(* PLC project drill, Dassault Systèmes ControlBuild 2024x Refresh1 *)
(* stored: creationDateTime 2024-03-18T15:45:01-01:00 *)

FUNCTION_BLOCK clampingfunction
  VAR_INPUT
    acknowledgePB : BOOL := false;
    releasing : BOOL := false;
    clamping : BOOL := false;
    rightUnlocked : BOOL := false;
    rightLocked : BOOL := false;
    leftUnlocked : BOOL := false;
    leftLocked : BOOL := false;
    rightFault : BOOL := false;
    leftFault : BOOL := false;
  END_VAR
  VAR_IN_OUT
    clampingDuration : INT := 0;
    releasingDuration : INT := 0;
  END_VAR
  VAR_OUTPUT
    clampingOK : BOOL := false;
    releasingOK : BOOL := false;
    clampingFault : INT := 0;
    rightLocking : BOOL := false;
    leftLocking : BOOL := false;
  END_VAR


ACTION C_source_code:

END_ACTION
END_FUNCTION_BLOCK

FUNCTION_BLOCK actions
  VAR_INPUT
    autoMode : BOOL := false;
    manualMode : BOOL := false;
    autoFwdCmd : BOOL := false;
    autoBwdCmd : BOOL := false;
    autoHSCmd : BOOL := false;
    autoLSCmd : BOOL := false;
    forwardPB : BOOL := false;
    backwardPB : BOOL := false;
    highSpeedPB : BOOL := false;
    lowSpeedPB : BOOL := false;
    stopPB : BOOL := false;
    generalFault : BOOL := false;
    autoWorkCmd : Unknown := ();
    valveWorkPB : Unknown := ();
  END_VAR
  VAR_OUTPUT
    forwardCmd : BOOL := false;
    backwardCmd : BOOL := false;
    highSpeedCmd : BOOL := false;
    lowSpeedCmd : BOOL := false;
    workCmd : BOOL := false;
  END_VAR


ACTION C_source_code:

END_ACTION
END_FUNCTION_BLOCK

FUNCTION_BLOCK faults1
  VAR_INPUT
    forwardCmd : BOOL := false;
    backwardCmd : BOOL := false;
    highSpeedCmd : BOOL := false;
    lowSpeedCmd : BOOL := false;
    thermalFB : BOOL := false;
    forwardFB : BOOL := false;
    backwardFB : BOOL := false;
    highSpeedFB : BOOL := false;
    lowSpeedFB : BOOL := false;
    acknowledgePB : BOOL := false;
    outletSensor : Unknown := ();
    inletSensor : Unknown := ();
    workCmd : Unknown := ();
  END_VAR
  VAR_IN_OUT
    thermalFault : BOOL := false;
    forwardFBFault : BOOL := false;
    backwardFBFault : BOOL := false;
  END_VAR
  VAR_OUTPUT
    generalFault : BOOL := false;
  END_VAR


ACTION C_source_code:

END_ACTION
END_FUNCTION_BLOCK

PROGRAM cmdofjack
  VAR_INPUT
    autoMode : BOOL := false;
    manualMode : BOOL := false;
    autoWorkCmd : BOOL := false;
    valveWorkPB : BOOL := false;
    outletSensor : BOOL := false;
    inletSensor : BOOL := false;
    acknowledgePB : BOOL := false;
  END_VAR
  VAR_OUTPUT
    workCmd : BOOL := false;
    generalFault : BOOL := false;
  END_VAR

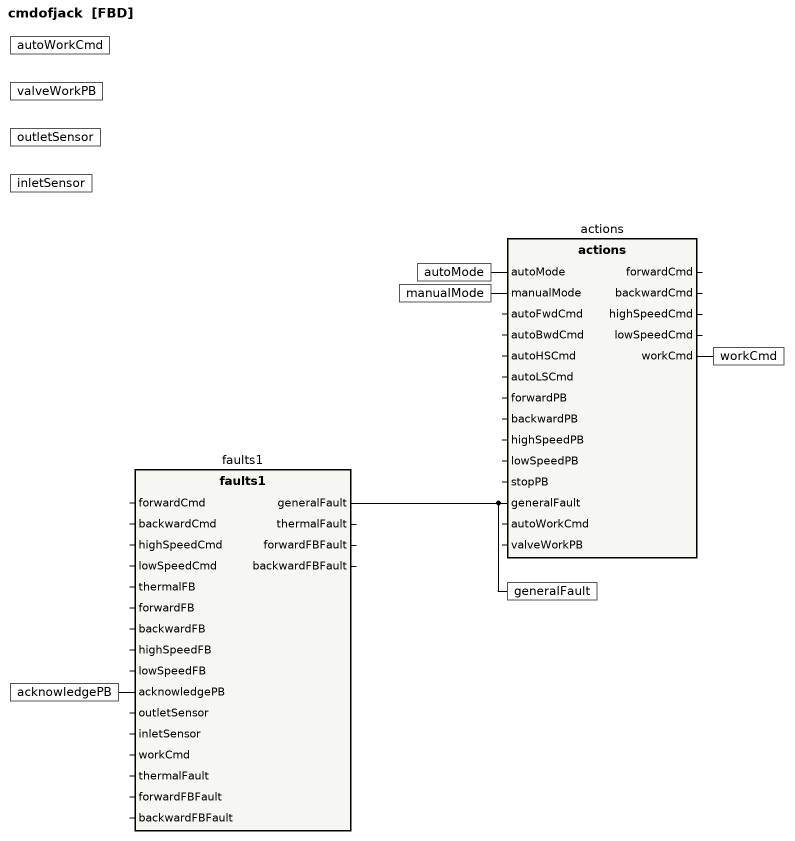
(* FBD diagram, written out as Structured Text *)
faults1(acknowledgePB := acknowledgePB);
actions(autoMode := autoMode, manualMode := manualMode, generalFault := faults1.generalFault);
workCmd := actions.workCmd;
generalFault := faults1.generalFault;
(* drawn but not wired to any output: autoWorkCmd, valveWorkPB, outletSensor, inletSensor *)
END_PROGRAM

FUNCTION_BLOCK jack
  VAR_INPUT
    energy : BOOL := false;
    cmdSupply : BOOL := false;
    sensorSupply : BOOL := false;
    valveWork : BOOL := false;
  END_VAR
  VAR_IN_OUT
    slidePosition : INT := 0;
    pipeWork : BOOL := false;
    pipeRest : BOOL := false;
    increment : REAL := 0.0;
    outletSensorLogic : BOOL := false;
    inletSensorLogic : BOOL := false;
    rodLength : REAL := 0.0;
    time2extend : REAL := 0.0;
    d_locking : BOOL := false;
    v_d_locking : REAL := 0.0;
    d_inletSensor : BOOL := false;
    v_d_inletSensor : BOOL := false;
    d_outletSensor : BOOL := false;
    v_d_outletSensor : BOOL := false;
  END_VAR
  VAR_OUTPUT
    outletSensor : BOOL := false;
    inletSensor : BOOL := false;
    rodPosition : REAL := 0.0;
    rodPercent : REAL := 0.0;
    incrementValue : REAL := 0.0;
  END_VAR


ACTION C_source_code:

END_ACTION
END_FUNCTION_BLOCK

FUNCTION_BLOCK backwardpb
  VAR_IN_OUT
    action : BOOL := false;
    timeCounter : REAL := 0.0;
    pulseDuration : REAL := 0.0;
    PBLogic : BOOL := false;
  END_VAR
  VAR_OUTPUT
    PB : BOOL := false;
  END_VAR


ACTION C_source_code:

END_ACTION
END_FUNCTION_BLOCK

FUNCTION_BLOCK forwardpb
  VAR_IN_OUT
    action : BOOL := false;
    timeCounter : REAL := 0.0;
    pulseDuration : REAL := 0.0;
    PBLogic : BOOL := false;
  END_VAR
  VAR_OUTPUT
    PB : BOOL := false;
  END_VAR


ACTION C_source_code:

END_ACTION
END_FUNCTION_BLOCK

FUNCTION_BLOCK speedswitch
  VAR_IN_OUT
    leftPosition : BOOL := false;
    rightPosition : BOOL := false;
  END_VAR
  VAR_OUTPUT
    leftVariable : BOOL := false;
    rightVariable : BOOL := false;
  END_VAR


ACTION C_source_code:

END_ACTION
END_FUNCTION_BLOCK

FUNCTION_BLOCK stoppb
  VAR_IN_OUT
    action : BOOL := false;
    timeCounter : REAL := 0.0;
    pulseDuration : REAL := 0.0;
    PBLogic : BOOL := false;
  END_VAR
  VAR_OUTPUT
    PB : BOOL := false;
  END_VAR


ACTION C_source_code:

END_ACTION
END_FUNCTION_BLOCK

PROGRAM panel1
  VAR_OUTPUT
    forwardPB : BOOL := false;
    backwardPB : BOOL := false;
    highSpeedPB : BOOL := false;
    lowSpeedPB : BOOL := false;
    stopPB : BOOL := false;
    valveWorkPB : BOOL := false;
  END_VAR

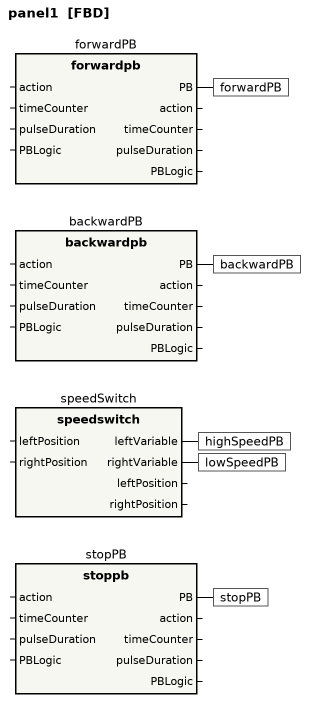
(* FBD diagram, written out as Structured Text *)
forwardPB();
forwardPB := forwardPB.PB;
backwardPB();
backwardPB := backwardPB.PB;
speedSwitch();
highSpeedPB := speedSwitch.leftVariable;
lowSpeedPB := speedSwitch.rightVariable;
stopPB();
stopPB := stopPB.PB;
END_PROGRAM

PROGRAM leftjack
  VAR_INPUT
    acknowledgePB : BOOL := false;
    autoMode : BOOL := false;
    manualMode : BOOL := false;
    autoWorkCmd : BOOL := false;
  END_VAR
  VAR_OUTPUT
    generalFault : BOOL := false;
    inletSensor : BOOL := false;
    outletSensor : BOOL := false;
    rodPosition : REAL := 0.0;
    rodPercent : REAL := 0.0;
    incrementValue : REAL := 0.0;
  END_VAR

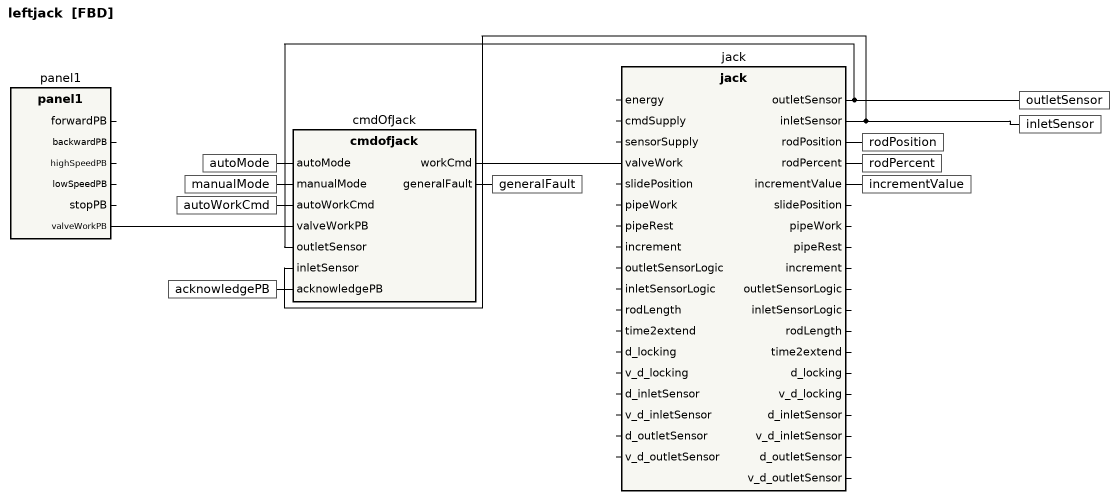
(* FBD diagram, written out as Structured Text *)
panel1();
jack(valveWork := cmdOfJack.workCmd);
cmdOfJack(autoMode := autoMode, manualMode := manualMode, autoWorkCmd := autoWorkCmd, valveWorkPB := panel1.valveWorkPB, outletSensor := jack.outletSensor, inletSensor := jack.inletSensor, acknowledgePB := acknowledgePB);
generalFault := cmdOfJack.generalFault;
inletSensor := jack.inletSensor;
outletSensor := jack.outletSensor;
rodPosition := jack.rodPosition;
rodPercent := jack.rodPercent;
incrementValue := jack.incrementValue;
END_PROGRAM

PROGRAM rightjack
  VAR_INPUT
    acknowledgePB : BOOL := false;
    autoMode : BOOL := false;
    manualMode : BOOL := false;
    autoWorkCmd : BOOL := false;
  END_VAR
  VAR_OUTPUT
    generalFault : BOOL := false;
    inletSensor : BOOL := false;
    outletSensor : BOOL := false;
    rodPosition : REAL := 0.0;
    rodPercent : REAL := 0.0;
    incrementValue : REAL := 0.0;
  END_VAR

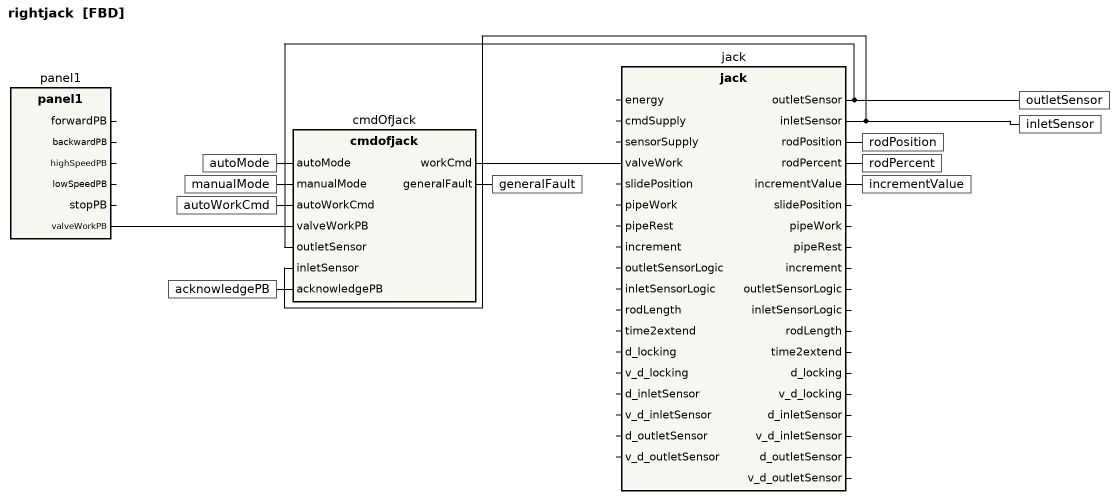
(* FBD diagram, written out as Structured Text *)
panel1();
jack(valveWork := cmdOfJack.workCmd);
cmdOfJack(autoMode := autoMode, manualMode := manualMode, autoWorkCmd := autoWorkCmd, valveWorkPB := panel1.valveWorkPB, outletSensor := jack.outletSensor, inletSensor := jack.inletSensor, acknowledgePB := acknowledgePB);
generalFault := cmdOfJack.generalFault;
inletSensor := jack.inletSensor;
outletSensor := jack.outletSensor;
rodPosition := jack.rodPosition;
rodPercent := jack.rodPercent;
incrementValue := jack.incrementValue;
END_PROGRAM

PROGRAM clamping
  VAR_INPUT
    acknowledgePB : BOOL := false;
    autoMode : BOOL := false;
    manualMode : BOOL := false;
    releasing : BOOL := false;
    clamping : BOOL := false;
  END_VAR
  VAR_OUTPUT
    clampingOK : BOOL := false;
    releasingOK : BOOL := false;
    clampingFault : INT := 0;
  END_VAR

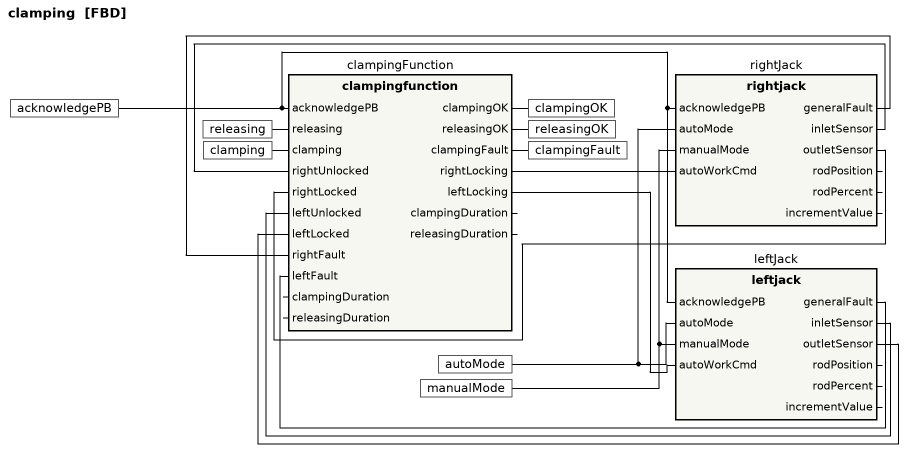
(* FBD diagram, written out as Structured Text *)
rightJack(acknowledgePB := acknowledgePB, autoMode := autoMode, manualMode := manualMode, autoWorkCmd := clampingFunction.rightLocking);
leftJack(acknowledgePB := acknowledgePB, autoMode := autoMode, manualMode := manualMode, autoWorkCmd := clampingFunction.leftLocking);
clampingFunction(acknowledgePB := acknowledgePB, releasing := releasing, clamping := clamping, rightUnlocked := rightJack.inletSensor, rightLocked := rightJack.outletSensor, leftUnlocked := leftJack.inletSensor, leftLocked := leftJack.outletSensor, rightFault := rightJack.generalFault, leftFault := leftJack.generalFault);
clampingOK := clampingFunction.clampingOK;
releasingOK := clampingFunction.releasingOK;
clampingFault := clampingFunction.clampingFault;
END_PROGRAM

FUNCTION_BLOCK ascentfunction
  VAR_INPUT
    acknowledgePB : BOOL := false;
    slowAscent : BOOL := false;
    fastAscent : BOOL := false;
    slowDescent : BOOL := false;
    fastDescent : BOOL := false;
    equipmentFault : BOOL := false;
  END_VAR
  VAR_OUTPUT
    motorFault : INT := 0;
    forward : BOOL := false;
    backward : BOOL := false;
    highSpeed : BOOL := false;
    lowSpeed : BOOL := false;
  END_VAR


ACTION C_source_code:

END_ACTION
END_FUNCTION_BLOCK

PROGRAM cmdofmotor
  VAR_INPUT
    autoMode : BOOL := false;
    manualMode : BOOL := false;
    autoFwdCmd : BOOL := false;
    autoBwdCmd : BOOL := false;
    autoHSCmd : BOOL := false;
    autoLSCmd : BOOL := false;
    forwardPB : BOOL := false;
    backwardPB : BOOL := false;
    highSpeedPB : BOOL := false;
    lowSpeedPB : BOOL := false;
    stopPB : BOOL := false;
    forwardFB : BOOL := false;
    backwardFB : BOOL := false;
    highSpeedFB : BOOL := false;
    lowSpeedFB : BOOL := false;
    thermalFB : BOOL := false;
    acknowledgePB : BOOL := false;
    autoCmd : Unknown := ();
  END_VAR
  VAR_OUTPUT
    forwardCmd : BOOL := false;
    backwardCmd : BOOL := false;
    highSpeedCmd : BOOL := false;
    lowSpeedCmd : BOOL := false;
    generalFault : BOOL := false;
  END_VAR

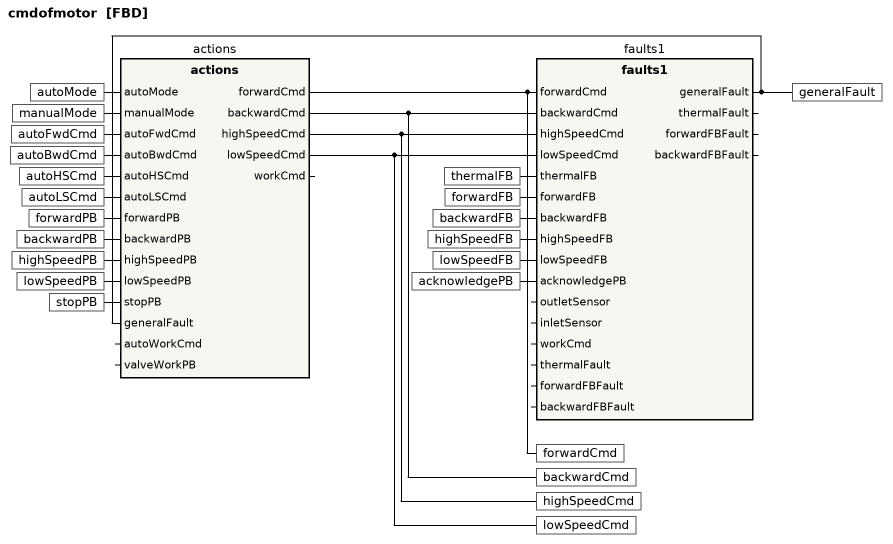
(* FBD diagram, written out as Structured Text *)
faults1(forwardCmd := actions.forwardCmd, backwardCmd := actions.backwardCmd, highSpeedCmd := actions.highSpeedCmd, lowSpeedCmd := actions.lowSpeedCmd, thermalFB := thermalFB, forwardFB := forwardFB, backwardFB := backwardFB, highSpeedFB := highSpeedFB, lowSpeedFB := lowSpeedFB, acknowledgePB := acknowledgePB);
actions(autoMode := autoMode, manualMode := manualMode, autoFwdCmd := autoFwdCmd, autoBwdCmd := autoBwdCmd, autoHSCmd := autoHSCmd, autoLSCmd := autoLSCmd, forwardPB := forwardPB, backwardPB := backwardPB, highSpeedPB := highSpeedPB, lowSpeedPB := lowSpeedPB, stopPB := stopPB, generalFault := faults1.generalFault);
forwardCmd := actions.forwardCmd;
backwardCmd := actions.backwardCmd;
highSpeedCmd := actions.highSpeedCmd;
lowSpeedCmd := actions.lowSpeedCmd;
generalFault := faults1.generalFault;
END_PROGRAM

FUNCTION_BLOCK motor
  VAR_INPUT
    voltage380 : BOOL := false;
    cmdSupply : BOOL := false;
    sensorSupply : BOOL := false;
    forward : BOOL := false;
    backward : BOOL := false;
    highSpeed : BOOL := false;
    lowSpeed : BOOL := false;
  END_VAR
  VAR_IN_OUT
    increment : REAL := 0.0;
    memoFwd : BOOL := false;
    memoBwd : BOOL := false;
    memoHighSpeed : BOOL := false;
    memoLowSpeed : BOOL := false;
    FwdHsState : BOOL := false;
    FwdLsState : BOOL := false;
    BwdHsState : BOOL := false;
    BwdLsState : BOOL := false;
    wantedSpeed : REAL := 0.0;
    nominalTime : REAL := 0.0;
    thermalLogic : BOOL := false;
    fwdFbLogic : BOOL := false;
    bwdFbLogic : BOOL := false;
    highSpeedFbLogic : BOOL := false;
    lowSpeedFbLogic : BOOL := false;
    nominalLowSpeed : REAL := 0.0;
    nominalHighSpeed : REAL := 0.0;
    d_locking : BOOL := false;
    v_d_locking : REAL := 0.0;
    d_electrical : BOOL := false;
    v_d_electrical : BOOL := false;
    d_forwardFB : BOOL := false;
    v_d_forwardFB : BOOL := false;
    d_highSpeedFB : BOOL := false;
    v_d_highSpeedFB : BOOL := false;
    d_lowSpeedFB : BOOL := false;
    v_d_lowSpeedFB : BOOL := false;
    d_backwardFB : BOOL := false;
    v_d_backwardFB : BOOL := false;
  END_VAR
  VAR_OUTPUT
    forwardFB : BOOL := false;
    backwardFB : BOOL := false;
    highSpeedFB : BOOL := false;
    lowSpeedFB : BOOL := false;
    thermal : BOOL := false;
    speedVal : REAL := 0.0;
    speedPercent : REAL := 0.0;
  END_VAR


ACTION C_source_code:

END_ACTION
END_FUNCTION_BLOCK

PROGRAM motorofturret
  VAR_INPUT
    autoMode : BOOL := false;
    manualMode : BOOL := false;
    autoFwdCmd : BOOL := false;
    autoBwdCmd : BOOL := false;
    autoHSCmd : BOOL := false;
    autoLSCmd : BOOL := false;
    acknowledgePB : BOOL := false;
  END_VAR
  VAR_OUTPUT
    speedVal : REAL := 0.0;
    speedPercent : REAL := 0.0;
    generalFault : BOOL := false;
  END_VAR

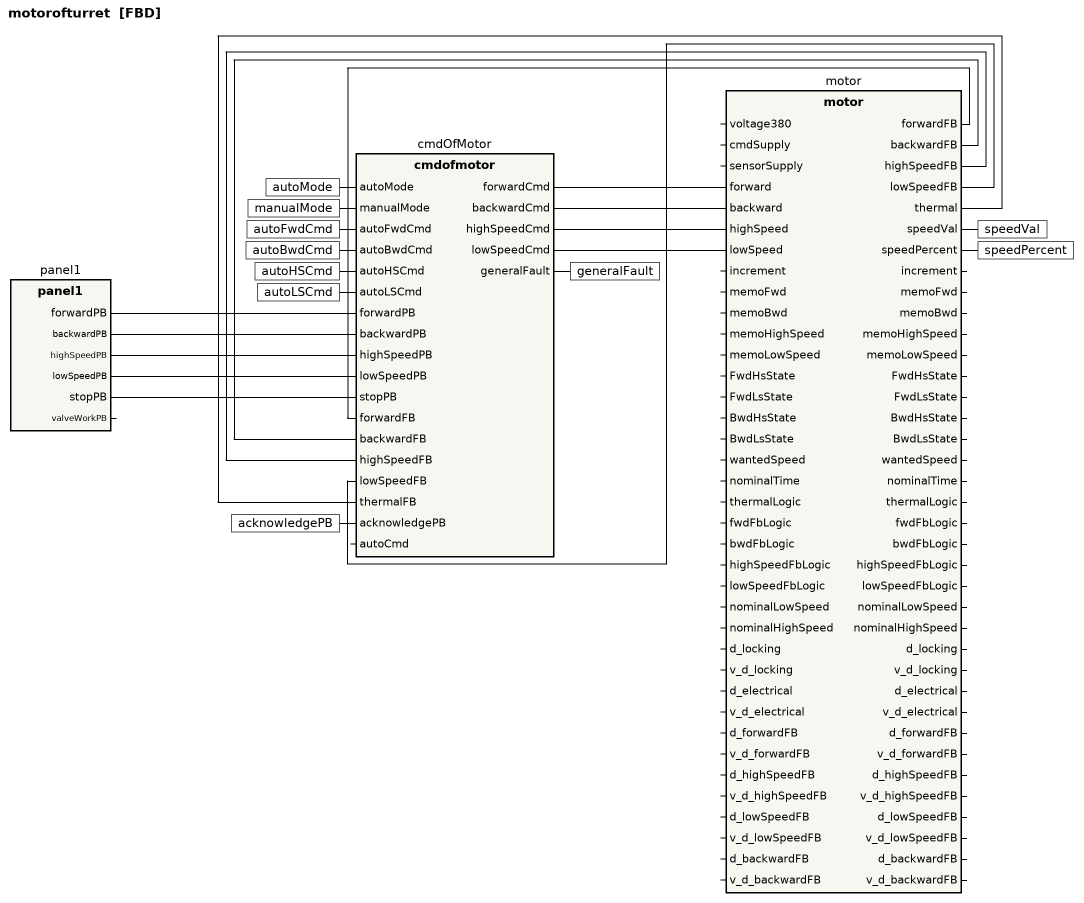
(* FBD diagram, written out as Structured Text *)
panel1();
cmdOfMotor(autoMode := autoMode, manualMode := manualMode, autoFwdCmd := autoFwdCmd, autoBwdCmd := autoBwdCmd, autoHSCmd := autoHSCmd, autoLSCmd := autoLSCmd, forwardPB := panel1.forwardPB, backwardPB := panel1.backwardPB, highSpeedPB := panel1.highSpeedPB, lowSpeedPB := panel1.lowSpeedPB, stopPB := panel1.stopPB, forwardFB := motor.forwardFB, backwardFB := motor.backwardFB, highSpeedFB := motor.highSpeedFB, lowSpeedFB := motor.lowSpeedFB, thermalFB := motor.thermal, acknowledgePB := acknowledgePB);
motor(forward := cmdOfMotor.forwardCmd, backward := cmdOfMotor.backwardCmd, highSpeed := cmdOfMotor.highSpeedCmd, lowSpeed := cmdOfMotor.lowSpeedCmd);
speedVal := motor.speedVal;
speedPercent := motor.speedPercent;
generalFault := cmdOfMotor.generalFault;
END_PROGRAM

FUNCTION_BLOCK turret
  VAR_INPUT
    speed : REAL := 0.0;
    forward : BOOL := false;
    backward : BOOL := false;
    highSpeed : BOOL := false;
    lowSpeed : BOOL := false;
  END_VAR
  VAR_IN_OUT
    speedIncrement : REAL := 0.0;
    lockingFault : BOOL := false;
    forwardEndFault : BOOL := false;
    forwardEndValue : BOOL := false;
    forwardDecelerationFault : BOOL := false;
    forwardDecelerationValue : BOOL := false;
    backwardDecelerationFault : BOOL := false;
    backwardDecelerationValue : BOOL := false;
    backwardEndFault : BOOL := false;
    backwardEndValue : BOOL := false;
    axleLength : REAL := 0.0;
    forwardDecelerationPosition : INT := 0;
    backwardDecelerationPosition : INT := 0;
    range : INT := 0;
  END_VAR
  VAR_OUTPUT
    axlePosition : REAL := 0.0;
    forwardEnd : BOOL := false;
    forwardDeceleration : BOOL := false;
    backwardDeceleration : BOOL := false;
    backwardEnd : BOOL := false;
  END_VAR


ACTION C_source_code:

END_ACTION
END_FUNCTION_BLOCK

PROGRAM descent
  VAR_INPUT
    slowAscent : BOOL := false;
    fastAscent : BOOL := false;
    slowDescent : BOOL := false;
    fastDescent : BOOL := false;
    acknowledgePB : BOOL := false;
    autoMode : BOOL := false;
    manualMode : BOOL := false;
  END_VAR
  VAR_OUTPUT
    ascentEnd : BOOL := false;
    topDeceleration : BOOL := false;
    downDeceleration : BOOL := false;
    descentEnd : BOOL := false;
    motorFault : INT := 0;
  END_VAR

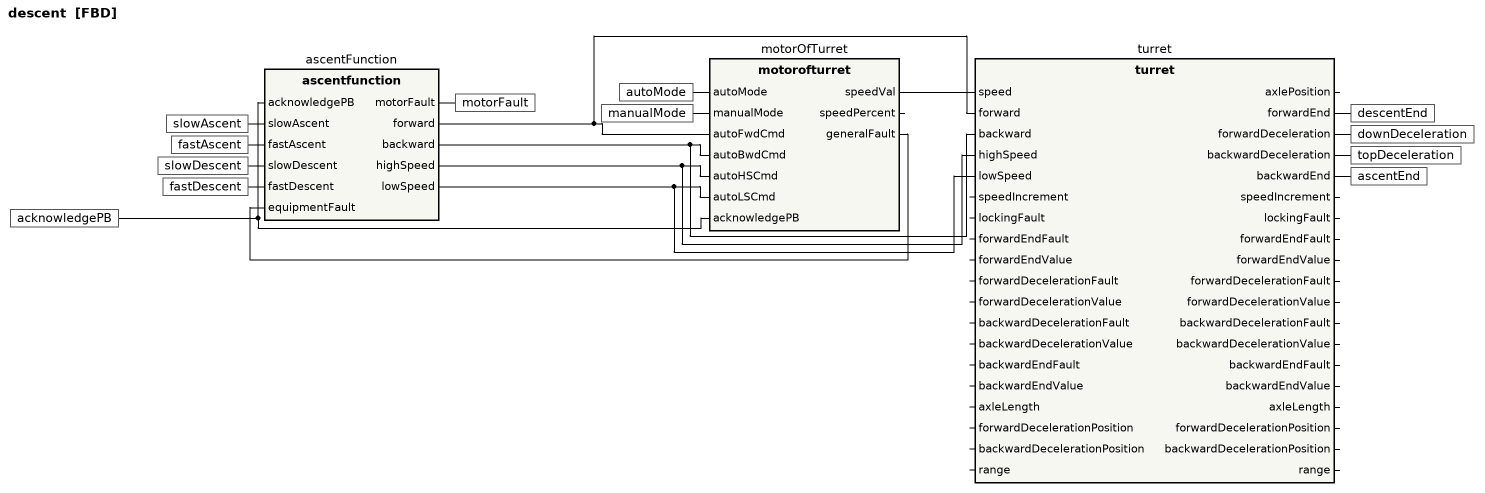
(* FBD diagram, written out as Structured Text *)
ascentFunction(acknowledgePB := acknowledgePB, slowAscent := slowAscent, fastAscent := fastAscent, slowDescent := slowDescent, fastDescent := fastDescent, equipmentFault := motorOfTurret.generalFault);
motorOfTurret(autoMode := autoMode, manualMode := manualMode, autoFwdCmd := ascentFunction.forward, autoBwdCmd := ascentFunction.backward, autoHSCmd := ascentFunction.highSpeed, autoLSCmd := ascentFunction.lowSpeed, acknowledgePB := acknowledgePB);
turret(speed := motorOfTurret.speedVal, forward := ascentFunction.forward, backward := ascentFunction.backward, highSpeed := ascentFunction.highSpeed, lowSpeed := ascentFunction.lowSpeed);
ascentEnd := turret.backwardEnd;
topDeceleration := turret.backwardDeceleration;
downDeceleration := turret.forwardDeceleration;
descentEnd := turret.forwardEnd;
motorFault := ascentFunction.motorFault;
END_PROGRAM

FUNCTION_BLOCK functionchart
  VAR_INPUT
    rotationFault : INT := 0;
    downState : BOOL := false;
    downDeceleration : BOOL := false;
    topDeceleration : BOOL := false;
    topState : BOOL := false;
    motorFault : INT := 0;
    clampingFault : INT := 0;
    releasingOK : BOOL := false;
    clampingOK : BOOL := false;
    emptyProd : BOOL := false;
    unitProd : BOOL := false;
    batchProd : BOOL := false;
    acknowledgePB : BOOL := false;
    piece : BOOL := false;
  END_VAR
  VAR_IN_OUT
    initialCond : BOOL := false;
    noFaultCond : BOOL := false;
    cnt : INT := 0;
    fastDescentDuration : INT := 0;
    slowDescentDuration : INT := 0;
    fastAscentDuration : INT := 0;
    slowAscentDuration : INT := 0;
  END_VAR
  VAR_OUTPUT
    rotation : BOOL := false;
    cycleEnd : BOOL := false;
    movementFault : INT := 0;
    loadingRequest : BOOL := false;
    unloadingRequest : BOOL := false;
    faultyState : BOOL := false;
    slowAscent : BOOL := false;
    fastAscent : BOOL := false;
    slowDescent : BOOL := false;
    fastDescent : BOOL := false;
    releasing : BOOL := false;
    clamping : BOOL := false;
  END_VAR


ACTION C_source_code:

END_ACTION
END_FUNCTION_BLOCK

PROGRAM spindlemotor
  VAR_INPUT
    autoMode : BOOL := false;
    manualMode : BOOL := false;
    autoCmd : BOOL := false;
    acknowledgePB : BOOL := false;
  END_VAR
  VAR_OUTPUT
    speedVal : REAL := 0.0;
    speedPercent : REAL := 0.0;
    generalFault : BOOL := false;
  END_VAR

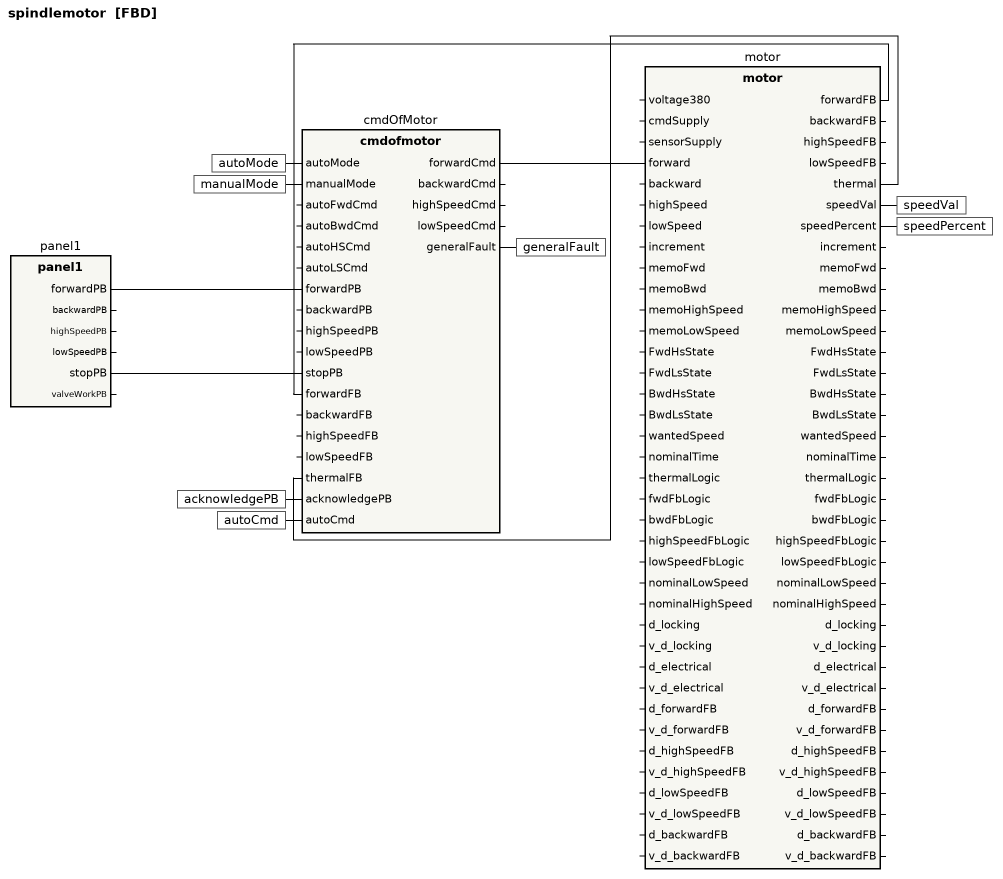
(* FBD diagram, written out as Structured Text *)
panel1();
cmdOfMotor(autoMode := autoMode, manualMode := manualMode, forwardPB := panel1.forwardPB, stopPB := panel1.stopPB, forwardFB := motor.forwardFB, thermalFB := motor.thermal, acknowledgePB := acknowledgePB, autoCmd := autoCmd);
motor(forward := cmdOfMotor.forwardCmd);
speedVal := motor.speedVal;
speedPercent := motor.speedPercent;
generalFault := cmdOfMotor.generalFault;
END_PROGRAM

PROGRAM spindle
  VAR_INPUT
    rotationFunction : BOOL := false;
    acknowledgePB : BOOL := false;
    autoMode : BOOL := false;
    manualMode : BOOL := false;
    rotation : Unknown := ();
    equipmentFault : Unknown := ();
  END_VAR
  VAR_OUTPUT
    rotationFault : INT := 0;
    contactor : BOOL := false;
  END_VAR

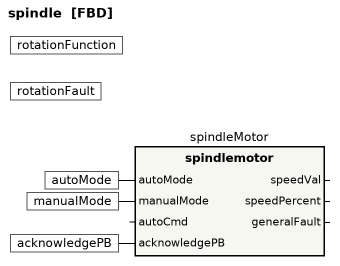
(* FBD diagram, written out as Structured Text *)
spindleMotor(autoMode := autoMode, manualMode := manualMode, acknowledgePB := acknowledgePB);
(* drawn but not wired to any output: rotationFunction *)
END_PROGRAM

PROGRAM functional
  VAR_INPUT
    piece : BOOL := false;
    emptyProd : BOOL := false;
    unitProd : BOOL := false;
    batchProd : BOOL := false;
    acknowledgePB : BOOL := false;
    autoMode : BOOL := false;
    manualMode : BOOL := false;
  END_VAR
  VAR_OUTPUT
    faultyState : BOOL := false;
    cycleEnd : BOOL := false;
    loadingRequest : BOOL := false;
    unloadingRequest : BOOL := false;
  END_VAR

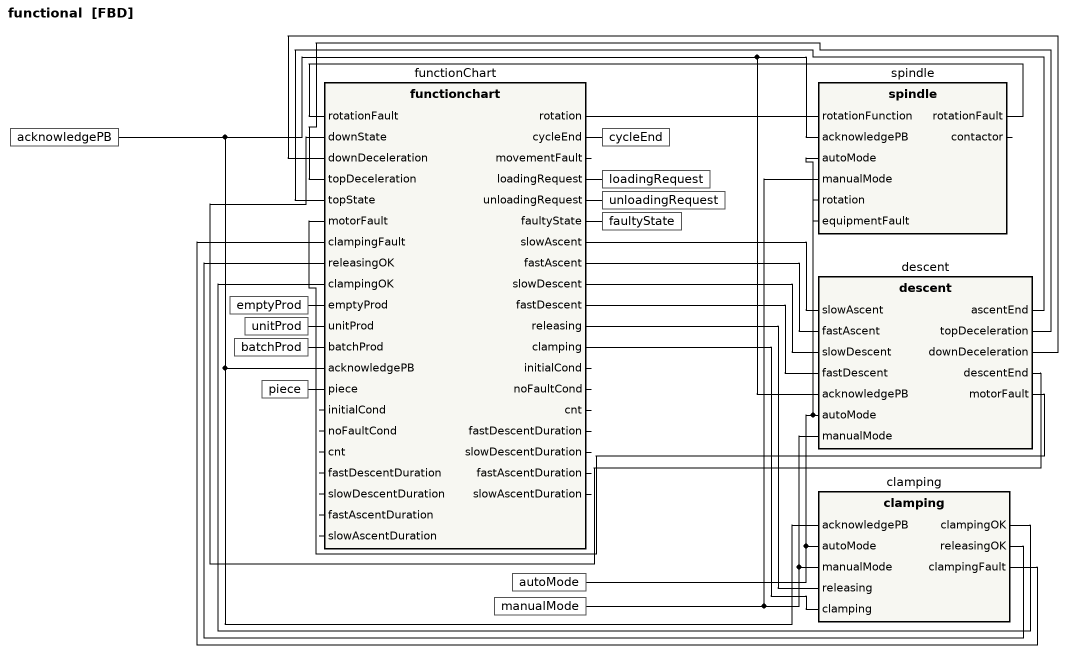
(* FBD diagram, written out as Structured Text *)
spindle(rotationFunction := functionChart.rotation, acknowledgePB := acknowledgePB, autoMode := autoMode, manualMode := manualMode);
descent(slowAscent := functionChart.slowAscent, fastAscent := functionChart.fastAscent, slowDescent := functionChart.slowDescent, fastDescent := functionChart.fastDescent, acknowledgePB := acknowledgePB, autoMode := autoMode, manualMode := manualMode);
clamping(acknowledgePB := acknowledgePB, autoMode := autoMode, manualMode := manualMode, releasing := functionChart.releasing, clamping := functionChart.clamping);
functionChart(rotationFault := spindle.rotationFault, downState := descent.descentEnd, downDeceleration := descent.downDeceleration, topDeceleration := descent.topDeceleration, topState := descent.ascentEnd, motorFault := descent.motorFault, clampingFault := clamping.clampingFault, releasingOK := clamping.releasingOK, clampingOK := clamping.clampingOK, emptyProd := emptyProd, unitProd := unitProd, batchProd := batchProd, acknowledgePB := acknowledgePB, piece := piece);
faultyState := functionChart.faultyState;
cycleEnd := functionChart.cycleEnd;
loadingRequest := functionChart.loadingRequest;
unloadingRequest := functionChart.unloadingRequest;
END_PROGRAM

FUNCTION_BLOCK acknowledgepb
  VAR_IN_OUT
    action : BOOL := false;
    timeCounter : REAL := 0.0;
    pulseDuration : REAL := 0.0;
    PBLogic : BOOL := false;
  END_VAR
  VAR_OUTPUT
    PB : BOOL := false;
  END_VAR


ACTION C_source_code:

END_ACTION
END_FUNCTION_BLOCK

FUNCTION_BLOCK cycleswitch
  VAR_IN_OUT
    leftPosition : BOOL := false;
    rightPosition : BOOL := false;
  END_VAR
  VAR_OUTPUT
    leftVariable : BOOL := false;
    rightVariable : BOOL := false;
  END_VAR


ACTION C_source_code:

END_ACTION
END_FUNCTION_BLOCK

FUNCTION_BLOCK emergencystop
  VAR_IN_OUT
    action : BOOL := false;
    PBLogic : BOOL := false;
  END_VAR
  VAR_OUTPUT
    pb : BOOL := false;
  END_VAR


ACTION C_source_code:

END_ACTION
END_FUNCTION_BLOCK

FUNCTION_BLOCK modeswitch
  VAR_IN_OUT
    leftPosition : BOOL := false;
    rightPosition : BOOL := false;
  END_VAR
  VAR_OUTPUT
    leftVariable : BOOL := false;
    rightVariable : BOOL := false;
  END_VAR


ACTION C_source_code:

END_ACTION
END_FUNCTION_BLOCK

FUNCTION_BLOCK poweruppb
  VAR_IN_OUT
    action : BOOL := false;
    timeCounter : REAL := 0.0;
    pulseDuration : REAL := 0.0;
    PBLogic : BOOL := false;
  END_VAR
  VAR_OUTPUT
    PB : BOOL := false;
  END_VAR


ACTION C_source_code:

END_ACTION
END_FUNCTION_BLOCK

FUNCTION_BLOCK startcyclepb
  VAR_IN_OUT
    action : BOOL := false;
    timeCounter : REAL := 0.0;
    pulseDuration : REAL := 0.0;
    PBLogic : BOOL := false;
  END_VAR
  VAR_OUTPUT
    PB : BOOL := false;
  END_VAR


ACTION C_source_code:

END_ACTION
END_FUNCTION_BLOCK

PROGRAM generalpanel
  VAR_OUTPUT
    powerUpPB : BOOL := false;
    startCyclePB : BOOL := false;
    emergencyStop : BOOL := false;
    batchCycle : BOOL := false;
    pieceCycle : BOOL := false;
    autoSwitch : BOOL := false;
    manualSwitch : BOOL := false;
    acknowledgePB : BOOL := false;
  END_VAR

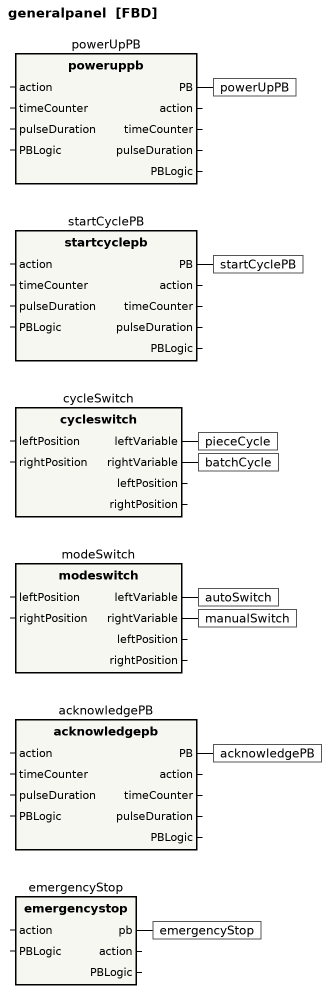
(* FBD diagram, written out as Structured Text *)
powerUpPB();
powerUpPB := powerUpPB.PB;
startCyclePB();
startCyclePB := startCyclePB.PB;
emergencyStop();
emergencyStop := emergencyStop.pb;
cycleSwitch();
batchCycle := cycleSwitch.rightVariable;
pieceCycle := cycleSwitch.leftVariable;
modeSwitch();
autoSwitch := modeSwitch.leftVariable;
manualSwitch := modeSwitch.rightVariable;
acknowledgePB();
acknowledgePB := acknowledgePB.PB;
END_PROGRAM

FUNCTION_BLOCK load
  VAR_INPUT
    loadingRequest : BOOL := false;
    unloadingRequest : BOOL := false;
  END_VAR
  VAR_IN_OUT
    count : INT := 0;
    loadingDuration : INT := 0;
  END_VAR
  VAR_OUTPUT
    piece : BOOL := false;
  END_VAR


ACTION C_source_code:

END_ACTION
END_FUNCTION_BLOCK

FUNCTION_BLOCK workingmodes
  VAR_INPUT
    powerUpPB : BOOL := false;
    startCyclePB : BOOL := false;
    emergencyStop : BOOL := false;
    batchCycle : BOOL := false;
    pieceCycle : BOOL := false;
    autoSwitch : BOOL := false;
    manualSwitch : BOOL := false;
    cycleEnd : BOOL := false;
    acknowledgePB : BOOL := false;
  END_VAR
  VAR_IN_OUT
    emergencyState : BOOL := false;
  END_VAR
  VAR_OUTPUT
    live : BOOL := false;
    autoMode : BOOL := false;
    manualMode : BOOL := false;
    emptyProd : BOOL := false;
    unitProd : BOOL := false;
    batchProd : BOOL := false;
  END_VAR


ACTION C_source_code:

END_ACTION
END_FUNCTION_BLOCK

PROGRAM my_app.drill

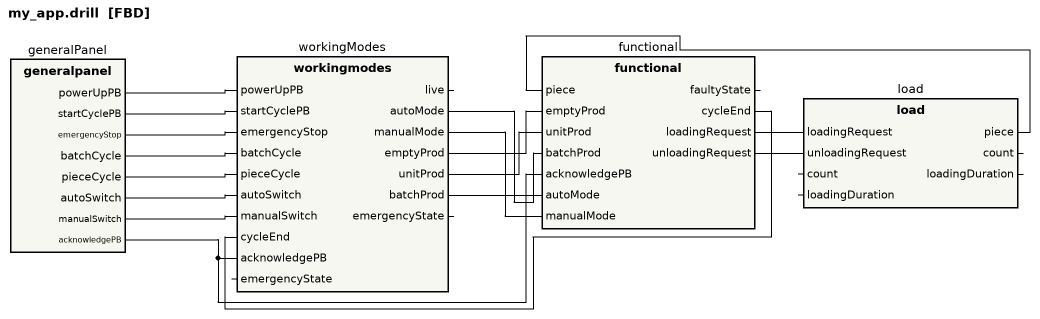
(* FBD diagram, written out as Structured Text *)
generalPanel();
load(loadingRequest := functional.loadingRequest, unloadingRequest := functional.unloadingRequest);
functional(piece := load.piece, emptyProd := workingModes.emptyProd, unitProd := workingModes.unitProd, batchProd := workingModes.batchProd, acknowledgePB := generalPanel.acknowledgePB, autoMode := workingModes.autoMode, manualMode := workingModes.manualMode);
workingModes(powerUpPB := generalPanel.powerUpPB, startCyclePB := generalPanel.startCyclePB, emergencyStop := generalPanel.emergencyStop, batchCycle := generalPanel.batchCycle, pieceCycle := generalPanel.pieceCycle, autoSwitch := generalPanel.autoSwitch, manualSwitch := generalPanel.manualSwitch, cycleEnd := functional.cycleEnd, acknowledgePB := generalPanel.acknowledgePB);
END_PROGRAM
